(* LS Electric XG5000 project: XMC_XYZ_Gantry *)
(* project for XYZ gantry example *)
(* PLC LSPLC *)
(* module base 0 slot 0: Input/Output Module:XMC-DN24 (DC 24V Input 8Points/TR output 16Points) *)
(* module base 0 slot 1: Internal Analog Input/Output:XMF-AH04E (A/D voltage/current 2 channels, D/A voltage 2 channels) *)
(* task Periodic Task: Kind=2 *)
(* task Initialization Task: Kind=1 *)
(* task NC Program: Kind=6 *)

PROGRAM GantryControl (* task: Scan Program *)
(* example program for gantry control. *)
VAR
    Enable_Gantry_Group : BOOL; (* command to enable the XYZ gantry group *)
    Enable_Power : BOOL; (* flag to enable all servo drives *)
    Execute_Connect : BOOL; (* flag to execute LS_Connect to connect EtherCAT network *)
    Execute_Disconnect : BOOL; (* flag to execute LS_Disconnect in cases where control must be disabled. *)
    Execute_GantryMove : BOOL; (* flag to execute an absolute position with linear interpolation *)
    Execute_GroupHome : BOOL; (* flag to execute the MC_GroupHome function *)
    Execute_GroupStop : BOOL; (* flag to execute stop for group motion *)
    Gantry_Group : UINT := 1; (* group to enable. *)
    Gantry_Velocity : LREAL; (* velocity in mm/second for gantry move *)
    Home_Position : ARRAY[0..9] OF LREAL; (* array of home positions for gantry initial values: Home_Position[6]=0, Home_Position[7]=0, Home_Position[4]=0, Home_Position[5]=0, Home_Position[2]=0, Home_Position[3]=0, Home_Position[0]=0, Home_Position[1]=0, Home_Position[8]=0, Home_Position[9]=0 *)
    INST_Connect : LS_CONNECT; (* LS_Connect FB *)
    INST_Disconnect : LS_DISCONNECT; (* LS_Disconnect FB *)
    INST_GroupEnable : MC_GROUPENABLE; (* function block to enable an Axis Group *)
    INST_GroupHome : MC_GROUPHOME; (* MC_GroupHome FB *)
    INST_GroupPower : MC_GROUPPOWER; (* Power on Axis Group *)
    INST_GroupStop : MC_GROUPSTOP; (* MC_GroupStop FB *)
    INST_MoveAbs : MC_MOVELINEARABSOLUTE; (* MC_MoveLinearAbsolute FB *)
    INST_PowerAll : MC_POWERALL; (* MC_PowerAll FB *)
    Move_Position : ARRAY[0..9] OF LREAL; (* array of positions for absolute linear interpolation move *)
END_VAR

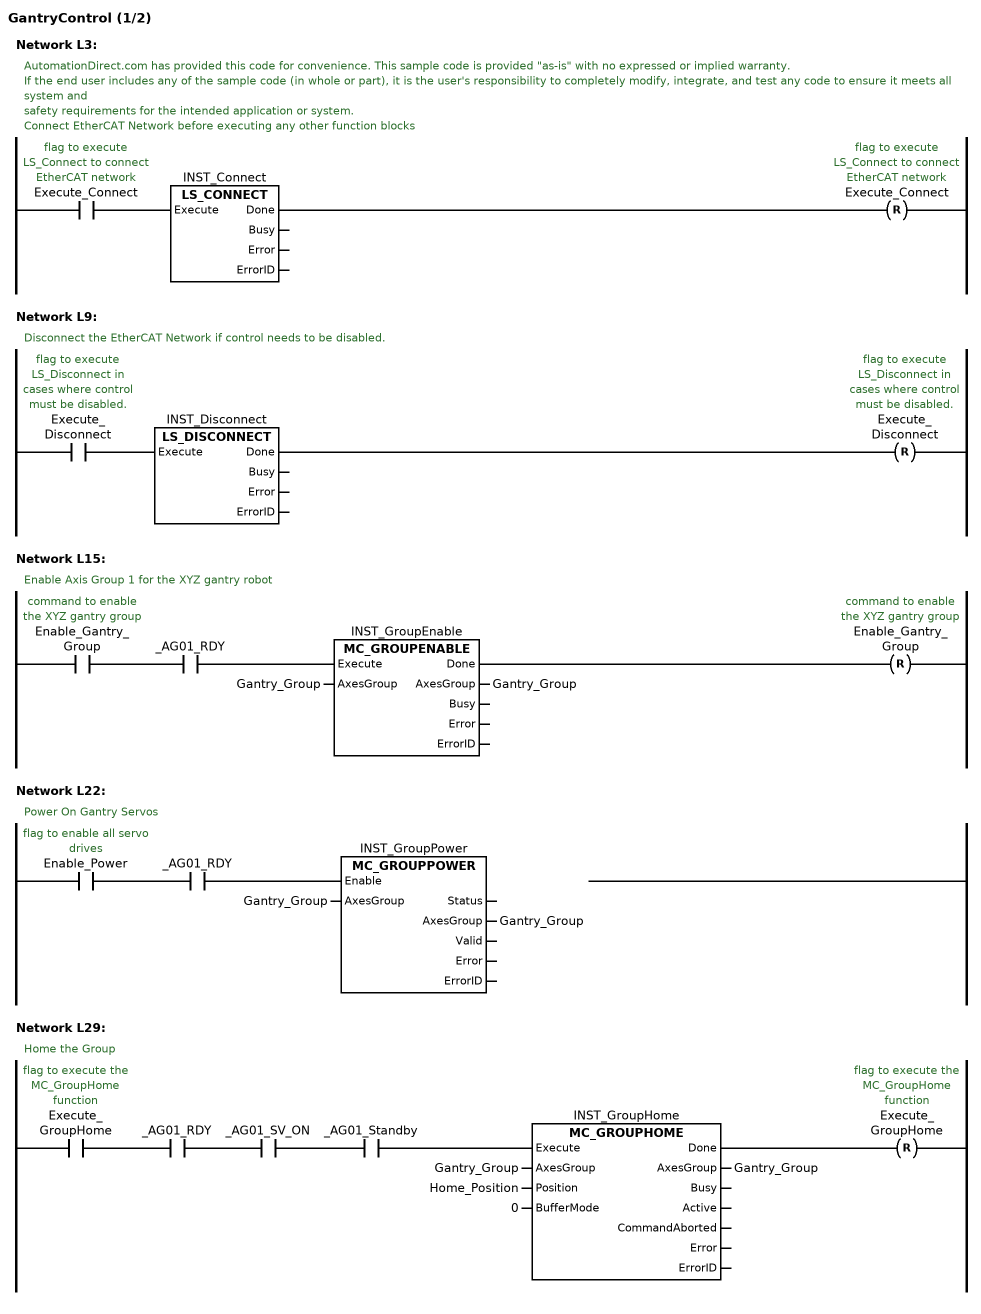
(* AutomationDirect.com has provided this code for convenience. This sample code is provided "as-is" with no expressed or implied warranty. / If the end user includes any of the sample code (in whole or part), it is the user's responsibility to completely modify, integrate, and test any code to ensure it meets all system and / safety requirements for the intended application or system. *)
(* Connect EtherCAT Network before executing any other function blocks *)
(* Rung L3 *)
INST_Connect(Execute := Execute_Connect);
IF INST_Connect.Done THEN Execute_Connect := FALSE; END_IF;
(* Disconnect the EtherCAT Network if control needs to be disabled. *)
(* Rung L9 *)
INST_Disconnect(Execute := Execute_Disconnect);
IF INST_Disconnect.Done THEN Execute_Disconnect := FALSE; END_IF;
(* Enable Axis Group 1 for the XYZ gantry robot *)
(* Rung L15 *)
INST_GroupEnable(Execute := Enable_Gantry_Group AND _AG01_RDY, AxesGroup := Gantry_Group, AxesGroup => Gantry_Group);
IF INST_GroupEnable.Done THEN Enable_Gantry_Group := FALSE; END_IF;
(* Power On Gantry Servos *)
(* Rung L22 *)
INST_GroupPower(Enable := Enable_Power AND _AG01_RDY, AxesGroup := Gantry_Group, AxesGroup => Gantry_Group);
(* Home the Group *)
(* Rung L29 *)
INST_GroupHome(Execute := Execute_GroupHome AND _AG01_RDY AND _AG01_SV_ON AND _AG01_Standby, AxesGroup := Gantry_Group, Position := Home_Position, BufferMode := 0, AxesGroup => Gantry_Group);
IF INST_GroupHome.Done THEN Execute_GroupHome := FALSE; END_IF;

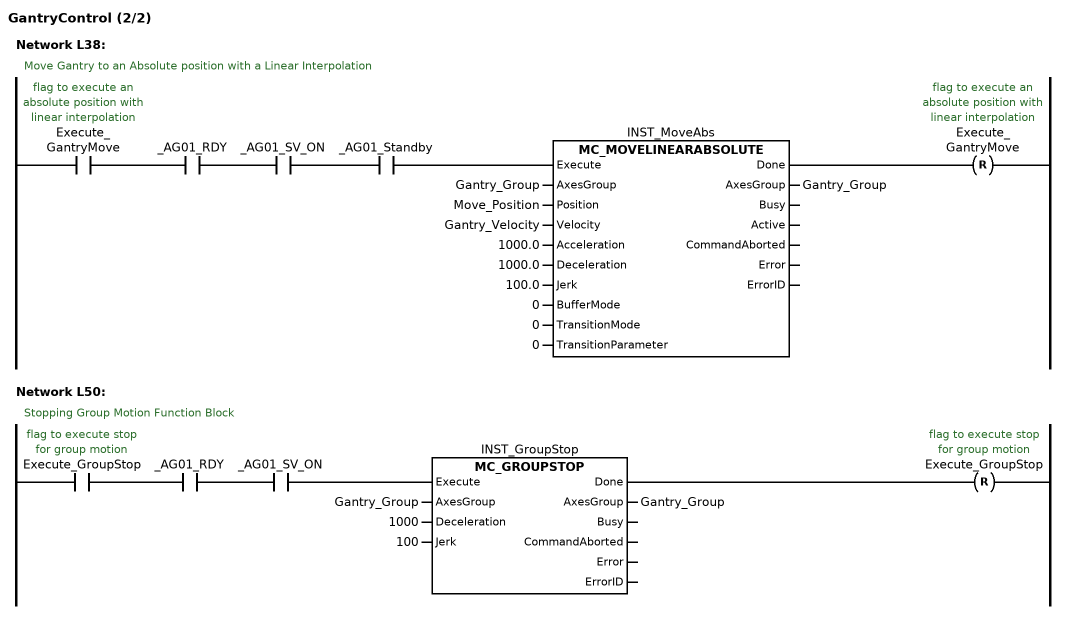
(* Move Gantry to an Absolute position with a Linear Interpolation *)
(* Rung L38 *)
INST_MoveAbs(Execute := Execute_GantryMove AND _AG01_RDY AND _AG01_SV_ON AND _AG01_Standby, AxesGroup := Gantry_Group, Position := Move_Position, Velocity := Gantry_Velocity, Acceleration := 1000.0, Deceleration := 1000.0, Jerk := 100.0, BufferMode := 0, TransitionMode := 0, TransitionParameter := 0, AxesGroup => Gantry_Group);
IF INST_MoveAbs.Done THEN Execute_GantryMove := FALSE; END_IF;
(* Stopping Group Motion Function Block *)
(* Rung L50 *)
INST_GroupStop(Execute := Execute_GroupStop AND _AG01_RDY AND _AG01_SV_ON, AxesGroup := Gantry_Group, Deceleration := 1000, Jerk := 100, AxesGroup => Gantry_Group);
IF INST_GroupStop.Done THEN Execute_GroupStop := FALSE; END_IF;
END_PROGRAM